TYPE Millimeter : LREAL;
END_TYPE

(* stored: Version 1.1.0.1, ProductVersion 3.1.4024.12
   DUT Millimeter: Id {a6b44fd6-3030-4d90-86ff-159d43ff61be} *)
